RoboDK station: New Station (1).rdk

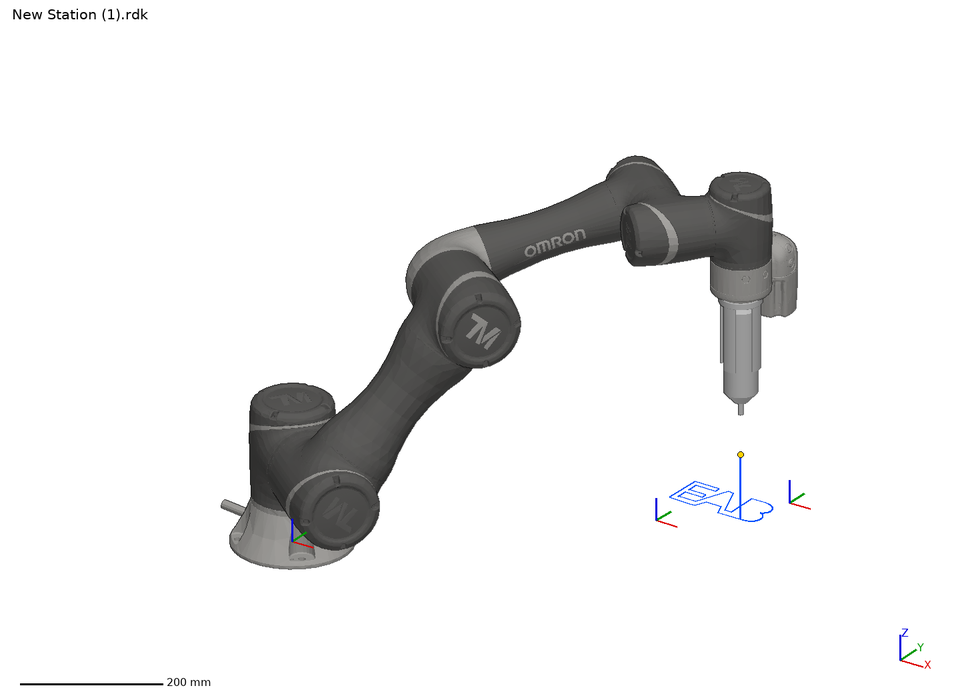
[picture v0: the station drawn from its stored meshes, robots at their saved joint values, targets as dots, program paths as lines]
Station New Station (1) (saved by RoboDK 5.6.7). Poses are relative to the parent item; angles as X-Y-Z fixed-axis rotations.
  - frame Omron TM5-700 Base at (0, 0, 0) mm
    - robot Omron TM5-700: 6 axes, payload 6 kg, reach 700 mm, repeatability 0.05 mm, weight 22.1 kg
        modified DH rows (alpha deg, a mm, theta deg, d mm): 0, 0, 0, 145.2; 90, 0, 90, 0; 0, 329, 0, 0; 0, 311, -90, 122.3; -90, 0, 0, 106.5; 90, 0, 180, 114.15
        joint limits [-270, -180, -155, -180, -180, -270] to [270, 180, 155, 180, 180, 270]; home [0, 0, 90, -90, 90, 0]; saved at [52.653, 39.424, 38.547, 12.028, 90, -37.347]
      - tool head true full 3, TCP at (0, 0, 250) mm, size 62.7 x 62.7 x 186 mm, geometry from head true full 3.stl
    - frame Reference Rhino at (500, 500, 0) mm
      - object Iost at (0, 0, 0) mm
  - frame Frame 2 at (379.33, 346.91, 0) mm
  - machining project Iost Settings: rotZ(0) | rotX(0)*rotY(0) | rotz(0) | 溙猱 | onStart | onPathStart | onApproach | onPoint | onRetract | onFinish | SetRPM(%1) | SetTool(%1) | Extruder(%1) | default | default | OutOnMov(%1) | OutOffMov(%1) | onPathFinish | M_RunCode(%1)
  - program Iost (120 instructions, listed below)
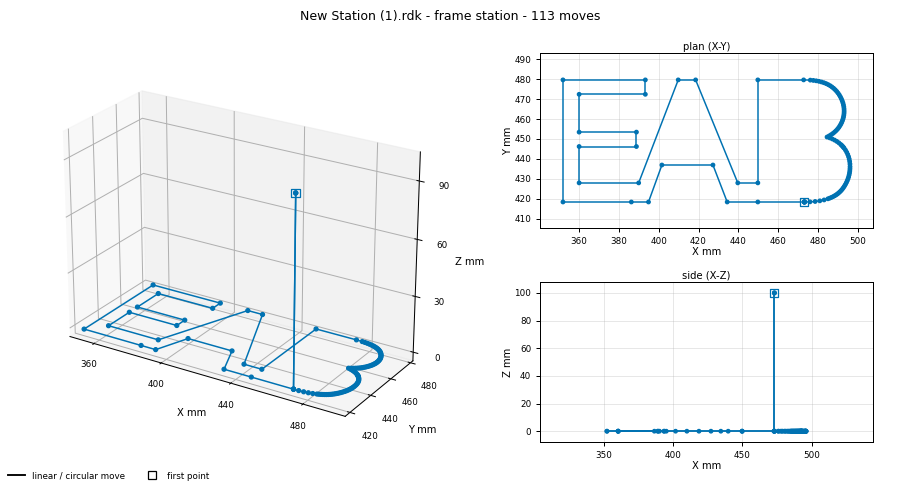
[picture p0: tool path of New Station (1).rdk in frame station, 113 of 113 moves have a stored position in this frame; points joined in program order, loops and branches not executed]

--- program Iost (robot Omron TM5-700) ---
  Smooth(1)
  Set speed (1000.0 mm/s)
  Set Ref.: Reference Rhino
  Set Tool: head true full 3
  Show head true full 3
  MoveJ 1 to (-26.89, -81.62, 100) mm, rotated rx 180 ry 0 rz 180 deg; joints [52.653, 39.424, 38.547, 12.028, 90, -37.347]
  MoveL 2 to (-26.89, -81.62, 100) mm, rotated rx 180 ry 0 rz 180 deg; joints [52.653, 39.424, 38.547, 12.028, 90, -37.347]
  MoveL 3 to (-26.89, -81.62, 0) mm, rotated rx 180 ry 0 rz 180 deg; joints [52.653, 38.438, 58.719, -7.157, 90, -37.347]
  MoveL 4 to (-26.89, -81.62, 0) mm, rotated rx 180 ry 0 rz 180 deg; joints [52.653, 38.438, 58.719, -7.157, 90, -37.347]
  Set speed (50.0 mm/s)
  MoveL 5 to (-24.08, -81.56, 0) mm, rotated rx 180 ry 0 rz -180 deg; joints [52.45, 38.883, 57.977, -6.861, 90, -37.55]
  MoveL 6 to (-21.5, -81.37, 0) mm, rotated rx 180 ry 0 rz -180 deg; joints [52.273, 39.315, 57.255, -6.571, 90, -37.727]
  MoveL 7 to (-19.14, -81.05, 0) mm, rotated rx 180 ry 0 rz -180 deg; joints [52.12, 39.733, 56.554, -6.288, 90, -37.88]
  MoveL 8 to (-17.01, -80.6, 0) mm, rotated rx 180 ry 0 rz 180 deg; joints [51.992, 40.137, 55.876, -6.012, 90, -38.008]
  MoveL 9 to (-15.08, -80.03, 0) mm, rotated rx 180 ry 0 rz -180 deg; joints [51.886, 40.529, 55.213, -5.742, 90, -38.114]
  MoveL 10 to (-14.18, -79.69, 0) mm, rotated rx 180 ry 0 rz 180 deg; joints [51.84, 40.723, 54.885, -5.608, 90, -38.16]
  MoveL 11 to (-13.32, -79.33, 0) mm, rotated rx 180 ry 0 rz -180 deg; joints [51.799, 40.915, 54.56, -5.474, 90, -38.201]
  MoveL 12 to (-12.5, -78.94, 0) mm, rotated rx 180 ry 0 rz -180 deg; joints [51.763, 41.105, 54.237, -5.342, 90, -38.237]
  MoveL 13 to (-11.73, -78.51, 0) mm, rotated rx -180 ry 0 rz 180 deg; joints [51.731, 41.293, 53.917, -5.21, 90, -38.269]
  MoveL 14 to (-11, -78.06, 0) mm, rotated rx 180 ry 0 rz 180 deg; joints [51.705, 41.48, 53.599, -5.079, 90, -38.295]
  MoveL 15 to (-10.31, -77.57, 0) mm, rotated rx 180 ry 0 rz -180 deg; joints [51.683, 41.665, 53.284, -4.949, 90, -38.317]
  MoveL 16 to (-9.65, -77.04, 0) mm, rotated rx 180 ry 0 rz -180 deg; joints [51.666, 41.85, 52.967, -4.818, 90, -38.334]
  MoveL 17 to (-9.02, -76.46, 0) mm, rotated rx 180 ry 0 rz -180 deg; joints [51.655, 42.04, 52.643, -4.683, 90, -38.345]
  MoveL 18 to (-8.42, -75.83, 0) mm, rotated rx 180 ry 0 rz -180 deg; joints [51.647, 42.234, 52.311, -4.545, 90, -38.353]
  MoveL 19 to (-7.85, -75.14, 0) mm, rotated rx 180 ry 0 rz -180 deg; joints [51.645, 42.432, 51.972, -4.404, 90, -38.355]
  MoveL 20 to (-7.3, -74.4, 0) mm, rotated rx 180 ry 0 rz -180 deg; joints [51.648, 42.634, 51.625, -4.259, 90, -38.352]
  MoveL 21 to (-6.78, -73.61, 0) mm, rotated rx 180 ry 0 rz 180 deg; joints [51.655, 42.84, 51.27, -4.11, 90, -38.345]
  MoveL 22 to (-6.28, -72.76, 0) mm, rotated rx -180 ry 0 rz -180 deg; joints [51.667, 43.051, 50.908, -3.958, 90, -38.333]
  MoveL 23 to (-5.82, -71.87, 0) mm, rotated rx 180 ry 0 rz 180 deg; joints [51.684, 43.266, 50.536, -3.802, 90, -38.316]
  MoveL 24 to (-5.39, -70.93, 0) mm, rotated rx 180 ry 0 rz -180 deg; joints [51.706, 43.48, 50.166, -3.646, 90, -38.294]
  MoveL 25 to (-5.02, -69.98, 0) mm, rotated rx 180 ry 0 rz 180 deg; joints [51.733, 43.689, 49.805, -3.493, 90, -38.267]
  MoveL 26 to (-4.71, -69.01, 0) mm, rotated rx 180 ry 0 rz 180 deg; joints [51.765, 43.892, 49.453, -3.345, 90, -38.235]
  MoveL 27 to (-4.45, -68.02, 0) mm, rotated rx 180 ry 0 rz -180 deg; joints [51.801, 44.088, 49.111, -3.2, 90, -38.199]
  MoveL 28 to (-4.26, -67.01, 0) mm, rotated rx -180 ry 0 rz -180 deg; joints [51.843, 44.279, 48.78, -3.059, 90, -38.157]
  MoveL 29 to (-4.11, -65.98, 0) mm, rotated rx 180 ry 0 rz 180 deg; joints [51.889, 44.464, 48.458, -2.922, 90, -38.111]
  MoveL 30 to (-4.03, -64.93, 0) mm, rotated rx -180 ry 0 rz -180 deg; joints [51.94, 44.643, 48.146, -2.789, 90, -38.06]
  MoveL 31 to (-4, -63.87, 0) mm, rotated rx 180 ry 0 rz 180 deg; joints [51.996, 44.816, 47.845, -2.66, 90, -38.004]
  MoveL 32 to (-4.05, -62.55, 0) mm, rotated rx 180 ry 0 rz 180 deg; joints [52.071, 45.015, 47.496, -2.511, 90, -37.929]
  MoveL 33 to (-4.19, -61.28, 0) mm, rotated rx 180 ry 0 rz 180 deg; joints [52.149, 45.193, 47.185, -2.378, 90, -37.851]
  MoveL 34 to (-4.42, -60.06, 0) mm, rotated rx 180 ry 0 rz 180 deg; joints [52.232, 45.347, 46.915, -2.262, 90, -37.768]
  MoveL 35 to (-4.75, -58.87, 0) mm, rotated rx 180 ry 0 rz -180 deg; joints [52.318, 45.478, 46.684, -2.163, 90, -37.682]
  MoveL 36 to (-5.17, -57.74, 0) mm, rotated rx 180 ry 0 rz 180 deg; joints [52.408, 45.587, 46.495, -2.081, 90, -37.592]
  MoveL 37 to (-5.68, -56.64, 0) mm, rotated rx 180 ry 0 rz -180 deg; joints [52.502, 45.671, 46.346, -2.017, 90, -37.498]
  MoveL 38 to (-6.29, -55.6, 0) mm, rotated rx -180 ry 0 rz 180 deg; joints [52.601, 45.732, 46.239, -1.971, 90, -37.399]
  MoveL 39 to (-6.99, -54.59, 0) mm, rotated rx -180 ry 0 rz -180 deg; joints [52.703, 45.77, 46.173, -1.943, 90, -37.297]
  MoveL 40 to (-7.37, -54.11, 0) mm, rotated rx 180 ry 0 rz 180 deg; joints [52.755, 45.779, 46.156, -1.935, 90, -37.245]
  MoveL 41 to (-7.77, -53.65, 0) mm, rotated rx 180 ry 0 rz -180 deg; joints [52.808, 45.782, 46.151, -1.933, 90, -37.192]
  MoveL 42 to (-8.2, -53.2, 0) mm, rotated rx -180 ry 0 rz -180 deg; joints [52.861, 45.779, 46.157, -1.936, 90, -37.139]
  MoveL 43 to (-8.64, -52.77, 0) mm, rotated rx 180 ry 0 rz -180 deg; joints [52.915, 45.769, 46.174, -1.943, 90, -37.085]
  MoveL 44 to (-9.59, -51.97, 0) mm, rotated rx 180 ry 0 rz -180 deg; joints [53.024, 45.73, 46.243, -1.973, 90, -36.976]
  MoveL 45 to (-10.62, -51.24, 0) mm, rotated rx 180 ry 0 rz -180 deg; joints [53.134, 45.665, 46.357, -2.022, 90, -36.866]
  MoveL 46 to (-11.72, -50.58, 0) mm, rotated rx -180 ry 0 rz -180 deg; joints [53.247, 45.574, 46.516, -2.09, 90, -36.753]
  MoveL 47 to (-12.91, -49.99, 0) mm, rotated rx 180 ry 0 rz 180 deg; joints [53.362, 45.459, 46.719, -2.178, 90, -36.638]
  MoveL 48 to (-14.18, -49.48, 0) mm, rotated rx -180 ry 0 rz -180 deg; joints [53.478, 45.318, 46.967, -2.284, 90, -36.522]
  MoveL 49 to (-15.53, -49.04, 0) mm, rotated rx 180 ry 0 rz 180 deg; joints [53.597, 45.152, 47.257, -2.409, 90, -36.403]
  MoveL 50 to (-14.49, -48.48, 0) mm, rotated rx 180 ry 0 rz -180 deg; joints [53.552, 45.427, 46.774, -2.201, 90, -36.448]
  MoveL 51 to (-13.51, -47.89, 0) mm, rotated rx 180 ry 0 rz -180 deg; joints [53.514, 45.7, 46.295, -1.995, 90, -36.486]
  MoveL 52 to (-12.61, -47.25, 0) mm, rotated rx 180 ry 0 rz -180 deg; joints [53.484, 45.97, 45.82, -1.79, 90, -36.516]
  MoveL 53 to (-11.77, -46.57, 0) mm, rotated rx 180 ry 0 rz -180 deg; joints [53.46, 46.237, 45.35, -1.587, 90, -36.54]
  MoveL 54 to (-11, -45.85, 0) mm, rotated rx 180 ry 0 rz -180 deg; joints [53.443, 46.501, 44.884, -1.385, 90, -36.557]
  MoveL 55 to (-10.3, -45.09, 0) mm, rotated rx 180 ry 0 rz -180 deg; joints [53.434, 46.761, 44.423, -1.184, 90, -36.566]
  MoveL 56 to (-9.66, -44.28, 0) mm, rotated rx 180 ry 0 rz -180 deg; joints [53.431, 47.018, 43.968, -0.986, 90, -36.569]
  MoveL 57 to (-9.1, -43.44, 0) mm, rotated rx 180 ry 0 rz 180 deg; joints [53.435, 47.272, 43.517, -0.789, 90, -36.565]
  MoveL 58 to (-8.6, -42.56, 0) mm, rotated rx 180 ry 0 rz 180 deg; joints [53.446, 47.52, 43.075, -0.596, 90, -36.554]
  MoveL 59 to (-8.16, -41.68, 0) mm, rotated rx 180 ry 0 rz 180 deg; joints [53.462, 47.76, 42.648, -0.408, 90, -36.538]
  MoveL 60 to (-7.8, -40.77, 0) mm, rotated rx 180 ry 0 rz -180 deg; joints [53.483, 47.992, 42.234, -0.226, 90, -36.517]
  MoveL 61 to (-7.5, -39.86, 0) mm, rotated rx 180 ry 0 rz -180 deg; joints [53.509, 48.216, 41.834, -0.05, 90, -36.491]
  MoveL 62 to (-7.27, -38.92, 0) mm, rotated rx -180 ry 0 rz -180 deg; joints [53.541, 48.431, 41.45, 0.12, 90, -36.459]
  MoveL 63 to (-7.1, -37.98, 0) mm, rotated rx 180 ry 0 rz -180 deg; joints [53.578, 48.637, 41.08, 0.283, 90, -36.422]
  MoveL 64 to (-7, -37.02, 0) mm, rotated rx 180 ry 0 rz 180 deg; joints [53.62, 48.834, 40.726, 0.44, 90, -36.38]
  MoveL 65 to (-6.97, -36.04, 0) mm, rotated rx 180 ry 0 rz -180 deg; joints [53.667, 49.023, 40.387, 0.59, 90, -36.333]
  MoveL 66 to (-7, -34.99, 0) mm, rotated rx 180 ry 0 rz -180 deg; joints [53.723, 49.212, 40.045, 0.742, 90, -36.277]
  MoveL 67 to (-7.12, -33.96, 0) mm, rotated rx -180 ry 0 rz 180 deg; joints [53.784, 49.387, 39.732, 0.882, 90, -36.216]
  MoveL 68 to (-7.3, -32.93, 0) mm, rotated rx -180 ry 0 rz -180 deg; joints [53.849, 49.545, 39.446, 1.009, 90, -36.151]
  MoveL 69 to (-7.57, -31.91, 0) mm, rotated rx 180 ry 0 rz -180 deg; joints [53.918, 49.687, 39.189, 1.124, 90, -36.082]
  MoveL 70 to (-7.9, -30.91, 0) mm, rotated rx 180 ry 0 rz -180 deg; joints [53.992, 49.813, 38.962, 1.225, 90, -36.008]
  MoveL 71 to (-8.32, -29.91, 0) mm, rotated rx -180 ry 0 rz 180 deg; joints [54.071, 49.922, 38.764, 1.314, 90, -35.929]
  MoveL 72 to (-8.81, -28.93, 0) mm, rotated rx 180 ry 0 rz -180 deg; joints [54.154, 50.015, 38.596, 1.389, 90, -35.846]
  MoveL 73 to (-9.37, -27.96, 0) mm, rotated rx 180 ry 0 rz 180 deg; joints [54.242, 50.091, 38.459, 1.451, 90, -35.758]
  MoveL 74 to (-10, -27.03, 0) mm, rotated rx 180 ry 0 rz 180 deg; joints [54.332, 50.146, 38.358, 1.496, 90, -35.668]
  MoveL 75 to (-10.68, -26.15, 0) mm, rotated rx 180 ry 0 rz -180 deg; joints [54.423, 50.179, 38.3, 1.522, 90, -35.577]
  MoveL 76 to (-11.43, -25.34, 0) mm, rotated rx -180 ry 0 rz -180 deg; joints [54.515, 50.187, 38.284, 1.529, 90, -35.485]
  MoveL 77 to (-12.23, -24.6, 0) mm, rotated rx 180 ry 0 rz 180 deg; joints [54.608, 50.172, 38.312, 1.516, 90, -35.392]
  MoveL 78 to (-13.09, -23.91, 0) mm, rotated rx 180 ry 0 rz 180 deg; joints [54.702, 50.133, 38.383, 1.484, 90, -35.298]
  MoveL 79 to (-14.01, -23.29, 0) mm, rotated rx 180 ry 0 rz -180 deg; joints [54.797, 50.07, 38.496, 1.434, 90, -35.203]
  MoveL 80 to (-14.98, -22.73, 0) mm, rotated rx 180 ry 0 rz 180 deg; joints [54.892, 49.984, 38.652, 1.364, 90, -35.108]
  MoveL 81 to (-16.01, -22.24, 0) mm, rotated rx -180 ry 0 rz -180 deg; joints [54.989, 49.875, 38.85, 1.275, 90, -35.011]
  MoveL 82 to (-17.11, -21.8, 0) mm, rotated rx 180 ry 0 rz 180 deg; joints [55.088, 49.74, 39.093, 1.167, 90, -34.912]
  MoveL 83 to (-18.3, -21.42, 0) mm, rotated rx -180 ry 0 rz -180 deg; joints [55.19, 49.578, 39.386, 1.036, 90, -34.81]
  MoveL 84 to (-19.58, -21.1, 0) mm, rotated rx 180 ry 0 rz 180 deg; joints [55.296, 49.389, 39.727, 0.884, 90, -34.704]
  MoveL 85 to (-20.95, -20.84, 0) mm, rotated rx 180 ry 0 rz 180 deg; joints [55.405, 49.174, 40.115, 0.711, 90, -34.595]
  MoveL 86 to (-22.4, -20.64, 0) mm, rotated rx 180 ry 0 rz -180 deg; joints [55.518, 48.933, 40.549, 0.519, 90, -34.482]
  MoveL 87 to (-23.93, -20.49, 0) mm, rotated rx 180 ry 0 rz -180 deg; joints [55.634, 48.667, 41.026, 0.307, 90, -34.366]
  MoveL 88 to (-27.27, -20.38, 0) mm, rotated rx 180 ry 0 rz -180 deg; joints [55.878, 48.063, 42.108, -0.171, 90, -34.122]
  MoveL 89 to (-50.25, -20.38, 0) mm, rotated rx 180 ry 0 rz -180 deg; joints [57.56, 44.114, 49.067, -3.181, 90, -32.44]
  MoveL 90 to (-50.25, -72.04, 0) mm, rotated rx 180 ry 0 rz -180 deg; joints [54.939, 36.269, 62.294, -8.563, 90, -35.061]
  MoveL 91 to (-60.31, -72.04, 0) mm, rotated rx 180 ry 0 rz 180 deg; joints [55.723, 34.847, 64.602, -9.449, 90, -34.277]
  MoveL 92 to (-81.45, -20.38, 0) mm, rotated rx 180 ry 0 rz 180 deg; joints [59.967, 39.48, 56.979, -6.459, 90, -30.033]
  MoveL 93 to (-90.18, -20.38, 0) mm, rotated rx 180 ry 0 rz -180 deg; joints [60.666, 38.294, 58.958, -7.253, 90, -29.334]
  MoveL 94 to (-110.03, -72.04, 0) mm, rotated rx 180 ry 0 rz -180 deg; joints [59.853, 28.405, 74.686, -13.091, 90, -30.147]
  MoveL 95 to (-139.9, -72.04, 0) mm, rotated rx 180 ry 0 rz -180 deg; joints [62.552, 24.913, 79.886, -14.799, 90, -27.448]
  MoveL 96 to (-139.9, -53.8, 0) mm, rotated rx 180 ry 0 rz 180 deg; joints [63.41, 27.401, 76.2, -13.602, 90, -26.59]
  MoveL 97 to (-111.15, -53.8, 0) mm, rotated rx -180 ry 0 rz 180 deg; joints [60.854, 30.747, 71.092, -11.839, 90, -29.146]
  MoveL 98 to (-111.15, -46.57, 0) mm, rotated rx 180 ry 0 rz -180 deg; joints [61.199, 31.759, 69.512, -11.271, 90, -28.801]
  MoveL 99 to (-139.9, -46.57, 0) mm, rotated rx 180 ry 0 rz 180 deg; joints [63.738, 28.412, 74.675, -13.087, 90, -26.262]
  MoveL 100 to (-139.9, -27.61, 0) mm, rotated rx 180 ry 0 rz 180 deg; joints [64.564, 31.141, 70.478, -11.619, 90, -25.436]
  MoveL 101 to (-106.68, -27.61, 0) mm, rotated rx 180 ry 0 rz 180 deg; joints [61.695, 35.065, 64.25, -9.315, 90, -28.305]
  MoveL 102 to (-106.68, -20.38, 0) mm, rotated rx 180 ry 0 rz 180 deg; joints [62.018, 36.158, 62.474, -8.633, 90, -27.982]
  MoveL 103 to (-148, -20.38, 0) mm, rotated rx 180 ry 0 rz -180 deg; joints [65.588, 31.314, 70.209, -11.523, 90, -24.412]
  MoveL 104 to (-148, -81.62, 0) mm, rotated rx 180 ry 0 rz -180 deg; joints [62.85, 22.727, 83.04, -15.767, 90, -27.15]
  MoveL 105 to (-113.7, -81.62, 0) mm, rotated rx 180 ry 0 rz -180 deg; joints [59.685, 26.7, 77.249, -13.949, 90, -30.315]
  MoveL 106 to (-105.1, -81.62, 0) mm, rotated rx -180 ry 0 rz -180 deg; joints [58.927, 27.746, 75.682, -13.428, 90, -31.073]
  MoveL 107 to (-98.37, -63.07, 0) mm, rotated rx 180 ry 0 rz -180 deg; joints [59.303, 31.045, 70.629, -11.673, 90, -30.697]
  MoveL 108 to (-72.76, -63.07, 0) mm, rotated rx 180 ry 0 rz 180 deg; joints [57.187, 34.366, 65.375, -9.741, 90, -32.813]
  MoveL 109 to (-65.62, -81.62, 0) mm, rotated rx 180 ry 0 rz 180 deg; joints [55.625, 32.842, 67.807, -10.648, 90, -34.375]
  MoveL 110 to (-50.25, -81.62, 0) mm, rotated rx -180 ry 0 rz 180 deg; joints [54.414, 34.98, 64.387, -9.367, 90, -35.586]
  MoveL 111 to (-26.89, -81.62, 0) mm, rotated rx 180 ry 0 rz 180 deg; joints [52.653, 38.438, 58.719, -7.157, 90, -37.347]
  Set speed (1000.0 mm/s)
  MoveL 112 to (-26.89, -81.62, 0) mm, rotated rx 180 ry 0 rz 180 deg; joints [52.653, 38.438, 58.719, -7.157, 90, -37.347]
  MoveL 113 to (-26.89, -81.62, 100) mm, rotated rx 180 ry 0 rz 180 deg; joints [52.653, 39.424, 38.547, 12.028, 90, -37.347]
